(* CODESYS project DicoCollections  Filefifo Demo.ecp
   Title: DicoCollections
   Placeholder: WagoIO
   DocFormat: reStructuredText
   Version: 1.0.0.0
   Company: Dicomat

Project tree, tasks and I/O mapping:
  PFC100_17 : 750-8101 PFC100 2ETH, WAGO, order no. 0750-8101, version 5.13.2.22
    application Application
      libraries: ; WagoAppTime, 1.7.3.0 (WAGO); Util, * (System); DicoCollections, 1.0.0.0 (Dicomat)
      task PLC_Task (cyclic, interval t#50ms, priority 15) calls PLC_PRG
      POU/
        program PLC_PRG [FBD]
        program RingFifoFileProducer [ST]
        program RingFifoFileConsumer [ST]
      data type TFifoItem
      global variables GVL
      function RealToStr [ST]
      function DTToStr [ST]
      global variables PV
    Kbus : Kbus, WAGO, version 1.4.0.2
        unmapped channels: K-BUS diagnostics
      _4_DI_Generic : 075x-4DI, WAGO, order no. 075x-4DI, version 0.0.0.13
          settings: K-BUS Module slot index = 1
          input  IO_xDI01 : BOOL  // _IN._IN
          input  IO_xDI02 : BOOL  // _IN._IN
          unmapped channels: _IN
      _2AI_TC_K_Diagn : 0750-0469, WAGO, order no. 0750-0469, version 0.0.0.9
          settings: K-BUS Module slot index = 2
          input  IO_iAI01 : INT  // _IINT 1
          unmapped channels: _IINT 2
      _4AO_4_20mA : 0750-0555, WAGO, order no. 0750-0555, version 0.0.0.12
          settings: K-BUS Module slot index = 3
          unmapped channels: _QW 1, _QW 2, _QW 3, _QW 4
      _16_DO_Generic : 075x-16DO, WAGO, order no. 075x-16DO, version 0.0.0.13
          settings: K-BUS Module slot index = 4
          unmapped channels: _OUT
    MODBUS
      MODBUS : MODBUS, WAGO, order no. n/a, version 1.1.1.15
    Serial
*)

// PFC100_17/Application/TFifoItem
TYPE TFifoItem :
STRUCT
	stTimeStamp: STRING(19);
	wdIndex    : WORD;
	stValue    : STRING(7);
	stTimeDone : STRING(19);	
END_STRUCT
END_TYPE

// PFC100_17/Application/GVL
{attribute 'qualified_only'}
VAR_GLOBAL
	FifoDebugBuffer: ARRAY [1..60] OF TFifoItem;
	FifoDebug      : RingFIFO;  
END_VAR

// PFC100_17/Application/PV
{attribute 'qualified_only'}
VAR_GLOBAL PERSISTENT RETAIN
	(* En memor*)
	FifoFile         : DicoCollections.RingFifoFile;
	wdConsumerHDL    : WORD;


END_VAR

// PFC100_17/Application/POU/PLC_PRG
PROGRAM PLC_PRG
VAR
	stFifoFileName	: STRING:= '/media/sd/filefifo.dat';
	wdProducerDone	: WORD;
	wdError       	: WORD;
	wdConsumerDone	: WORD;
	(*....*)
	SimData			: Util.RAMP_REAL;
	rlTemperature	: REAL;
	rsSelect: rs;

	rlSetPointTemp : REAL:= 21;
	rlMaxTemp      : REAL:= 23;
	rlMinTemp      : REAL:= 18;
END_VAR

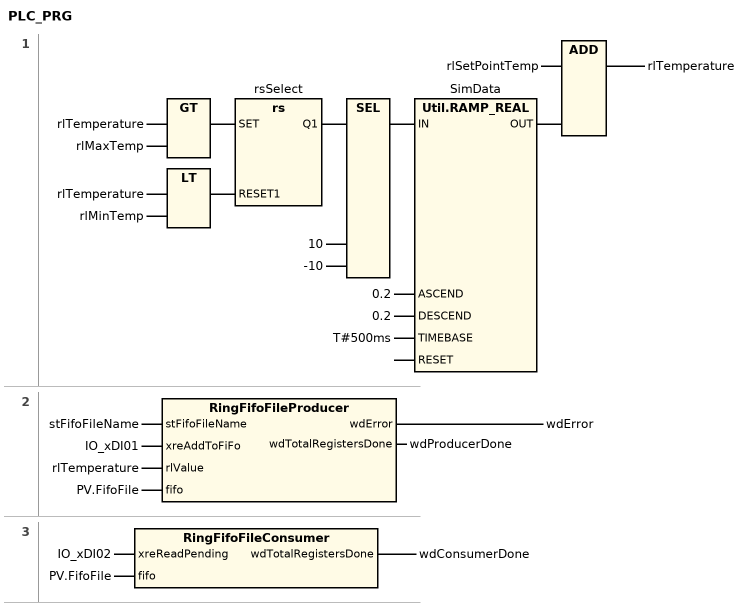
// NETWORK 1
rsSelect(SET := rlTemperature > rlMaxTemp, RESET1 := rlTemperature < rlMinTemp); // rs
SimData(IN := SEL(rsSelect.Q1, 10, -10), ASCEND := 0.2, DESCEND := 0.2, TIMEBASE := T#500ms); // Util.RAMP_REAL
rlTemperature := rlSetPointTemp + SimData.OUT;

// NETWORK 2
RingFifoFileProducer(stFifoFileName := stFifoFileName, xreAddToFiFo := IO_xDI01, rlValue := rlTemperature, fifo := PV.FifoFile, wdTotalRegistersDone => wdProducerDone);
wdError := RingFifoFileProducer.wdError;

// NETWORK 3
RingFifoFileConsumer(xreReadPending := IO_xDI02, fifo := PV.FifoFile);
wdConsumerDone := RingFifoFileConsumer.wdTotalRegistersDone;

END_PROGRAM

// PFC100_17/Application/POU/RingFifoFileProducer
PROGRAM RingFifoFileProducer
VAR CONSTANT
	_MAX_FIFO_ITEMS: WORD:= 10; (* Número máximo de *) 
END_VAR
VAR_INPUT
	stFifoFileName: STRING:= '/media/sd/filefifo.dat'; 
	xreAddToFiFo  : BOOL;
	rlValue       : REAL;
END_VAR
VAR_IN_OUT
	fifo: RingFifoFile;
END_VAR
VAR_OUTPUT
	wdError: WORD;
	wdTotalRegistersDone: WORD; 
END_VAR

VAR
	_FifoItem: TFifoItem;
	_rtgAddToFifo: R_TRIG;
	_wdOverWrittenEvents: WORD;
END_VAR

IF NOT fifo.Initialized THEN
	IF wdError = 0 THEN
		fifo.Init( stFifoFileName, _MAX_FIFO_ITEMS, SIZEOF(_FifoItem));	// ss	
	END_IF
END_IF
_rtgAddToFifo( CLK:= xreAddToFiFo);
IF fifo.Initialized THEN
	IF _rtgAddToFifo.Q THEN
		_FifoItem.stTimeStamp:= DTToStr(FuGetDateAndTime());
		_FifoItem.wdIndex:= _FifoItem.wdIndex + 1; 
		_FifoItem.stValue    := RealToStr(rlValue, 1);
		(* ++++++++ *)
		IF fifo.Push( ADR(_FifoItem)) > 0 THEN
			(* Se sobre-escriben clientes *)			
			_wdOverWrittenEvents:= _wdOverWrittenEvents + 1;
		END_IF
		(* *)
		wdTotalRegistersDone:= wdTotalRegistersDone + 1;
	END_IF 
END_IF

END_PROGRAM

// PFC100_17/Application/DTToStr
FUNCTION DTToStr: STRING(19)
VAR_INPUT
	dtDateTime: DT;
END_VAR
VAR
	_stdummy: STRING(22); 
END_VAR

_stdummy:= DT_TO_STRING(dtDateTime);
DTToStr:= RIGHT( _stdummy, 19);

END_FUNCTION

// PFC100_17/Application/RealToStr
FUNCTION RealToStr: STRING(25)
VAR_INPUT
	rlValue   : REAL;
	btDecimals: BYTE;
END_VAR
VAR
	_iLength: int;
	_iPosition: INT;
END_VAR

RealToStr:= REAL_TO_STRING(rlValue);
_iLength:= LEN(RealToStr);
_iPosition:= FIND(RealToStr, '.');
IF btDecimals > 0 THEN
	IF _iLength - _iPosition > btDecimals THEN
		RealToStr:= LEFT( RealToStr, _iPosition  + btDecimals);
	END_IF
ELSE
	IF _iPosition > 0 THEN
		RealToStr:= LEFT( RealToStr, _iPosition - 1);
	END_IF
END_IF

END_FUNCTION

// PFC100_17/Application/POU/RingFifoFileConsumer
PROGRAM RingFifoFileConsumer
VAR_INPUT
	xreReadPending: BOOL;
END_VAR
VAR_IN_OUT
	fifo: DicoCollections.RingFifoFile;
END_VAR
VAR_OUTPUT
	wdTotalRegistersDone: WORD; 
END_VAR
VAR
	_rtgReadAll: R_TRIG;
	_FifoItem: TFifoItem;
END_VAR

(* Para depuerar utilzamos un fifo en memoria *)
IF NOT( GVL.FifoDebug.Initialized) THEN
	GVL.FifoDebug.Init( ADR(GVL.FifoDebugBuffer), SIZEOF(GVL.FifoDebugBuffer), SIZEOF(GVL.FifoDebugBuffer[1])); 
END_IF 

(* *)
IF NOT( fifo.IsValidHandler(PV.wdConsumerHDL)) THEN
	PV.wdConsumerHDL:= fifo.Open();
END_IF
_rtgReadAll( CLK:= xreReadPending);
IF fifo.IsValidHandler(PV.wdConsumerHDL) THEN
	IF _rtgReadAll.Q THEN
		WHILE fifo.Pop( PV.wdConsumerHDL, ADR(_FifoItem), TRUE) DO 
			_FifoItem.stTimeDone:= DTToStr(FuGetDateAndTime());
			GVL.FifoDebug.Push( ADR(_FifoItem));
			wdTotalRegistersDone:= wdTotalRegistersDone + 1;
		END_WHILE
	END_IF
END_IF

END_PROGRAM
